///EL1002 | 2-channel digital input terminal 24 V DC, 3 ms
FUNCTION_BLOCK EL1002_v1_00
VAR_INPUT
	En: BOOL;
END_VAR
VAR_OUTPUT
	EnO: BOOL;
	bDi_1: BOOL;
	bDi_2: BOOL;
	bError: BOOL;
END_VAR
VAR
	Channel_1_Input AT %I*: BOOL;
	Channel_2_Input AT %I*: BOOL;
	WcState_WcState AT %I*: BOOL;
	InfoData_State AT %I*: UINT;
END_VAR

EnO:=En;

IF En AND (WcState_WcState OR InfoData_State<>16#8) THEN
	bError:=TRUE;
ELSE
	bError:=FALSE;
END_IF

IF En THEN
	IF bError=FALSE THEN
		bDi_1:=Channel_1_Input;
		bDi_2:=Channel_2_Input;
	ELSE
		bDi_1:=FALSE;
		bDi_2:=FALSE;
	END_IF
END_IF

END_FUNCTION_BLOCK

(* stored: Version 1.1.0.1, ProductVersion 3.1.0.25
   POU EL1002_v1_00: Id {c9bcbe69-7d2c-4bc2-8415-5240f6e73522} *)
